{attribute 'qualified_only'}
{attribute 'strict'}
{attribute 'to_string'}
TYPE E_Color :
(
	eSilver,
	eLime,
	eYellow,
	eOrange,
	eRed,
	eBlue
);
END_TYPE

(* stored: Version 1.1.0.1, ProductVersion 3.1.4026.17
   DUT E_Color: Id {2789594e-f701-4945-839b-81566fe8b622} *)
